GLOBALCONSTANTS storageStatusMessages (* Global constants for storage status messages (INI and NVS) *)
  (* Standard: 61499-1 *)
  (* Version 1.2, 2026-08-01, franz, added read-only settings error message *)
  (* Version 1.1, 2026-06-13, franz *)
  PACKAGE logiBUS::storage::const;
  VAR_GLOBAL CONSTANT
    OK : STRING := 'OK';
    NO_CHANGE : STRING := 'Value was not stored. Old is new';
    INITIALISED : STRING := 'initialized';
    NOT_INITIALISED : STRING := 'Not initialized';
    ERR : STRING := 'ERROR';
    ERR_NVS_NOT_FOUND : STRING := 'ESP_ERR_NVS_NOT_FOUND';
    ERR_NVS_DEFAULT_SET : STRING := 'Default Value was used';
    ERR_SECTION_EMPTY : STRING := 'SECTION empty';
    ERR_KEY_EMPTY : STRING := 'KEY empty';
    ERR_SECTION_WHITESPACE : STRING := 'SECTION contains whitespace';
    ERR_KEY_WHITESPACE : STRING := 'KEY contains whitespace';
    ERR_READ_ONLY : STRING := 'Key is read-only';
  END_VAR
END_GLOBALCONSTANTS
